// TIA Portal V18 export
FUNCTION "Pressure control" : Void   // FC24, LAD
{ S7_Optimized_Access := 'TRUE' }
VERSION : 0.1
// stored: AutoNumber true, IsIECCheckEnabled false, SetENOAutomatically false, UDAEnableTagReadback false
BEGIN

REGION Network 1 (SCL): Pump A pressure setting Inlet

   IF "Pressure sensor Pump Inlet A" < 32767 AND "Control".Pressure_sensor_select = 0 THEN
       "pressure".Misc."Pump A Scalx valueIN" := SCALE_X(MIN := 0.0,
                                                           VALUE := NORM_X(MIN := 0,
                                                                           VALUE := "Pressure sensor Pump Inlet A",
                                                                           MAX := 27648),
                                                           MAX := "pressure".A."pressure at 20mA");
   ELSIF "Pressure sensor Pump Inlet A_mA" < 32767 AND "Control".Pressure_sensor_select = 1 THEN
       "pressure".Misc."Pump A Scalx valueIN" := SCALE_X(MIN := 0.0,
                                                           VALUE := NORM_X(MIN := 0,
                                                                           VALUE := "Pressure sensor Pump Inlet A_mA",
                                                                           MAX := 27648),
                                                           MAX := "pressure".A."pressure at 20mA");
   END_IF;

   "Alarm_DB".input.alarm[15] := (("Control".Pressure_sensor_select = 0) AND ("Pressure sensor Pump Inlet A" >= 32767)) OR (("Control".Pressure_sensor_select = 1) AND ("Pressure sensor Pump Inlet A_mA" >= 32767));
END_REGION

REGION Network 2 (SCL): Pump A pressure setting Outlet

   IF "Pressure Sensor Pump Outlet A" < 32767 THEN
       "pressure".Misc."Pump A Scalx valueOUT" := SCALE_X(MIN := 0.0,
                                                           VALUE := NORM_X(MIN := 0,
                                                                           VALUE := "Pressure Sensor Pump Outlet A",
                                                                           MAX := 27648),
                                                           MAX := "pressure".A_Outlet."pressure at 20mA");
   END_IF;
END_REGION

REGION Network 3: gear Pump A pressure
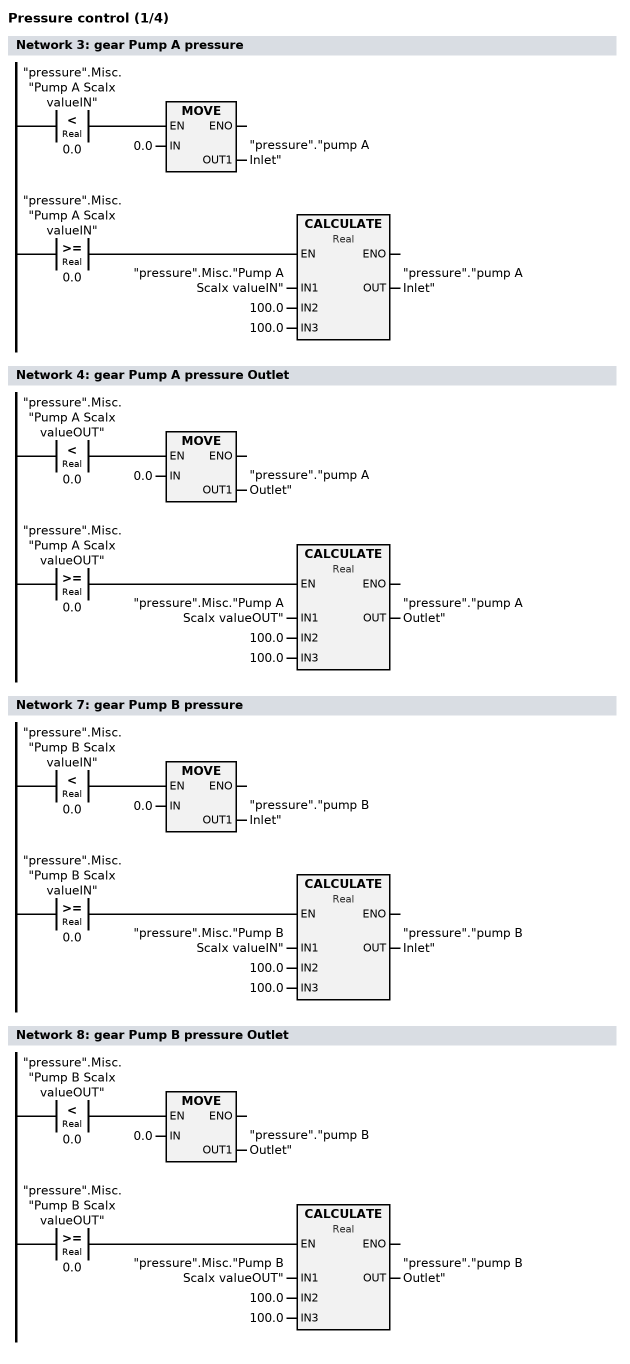
   RUNG wire#powerrail
      { S7_Templates := "SrcType := Real" } LT_Contact(in1 := "pressure".Misc."Pump A Scalx valueIN", in2 := 0.0)
      Move(in := 0.0, out1 => "pressure"."pump A Inlet")
   END_RUNG
   RUNG wire#powerrail
      { S7_Templates := "SrcType := Real" } GE_Contact(in1 := "pressure".Misc."Pump A Scalx valueIN", in2 := 0.0)
      { S7_Templates := "SrcType := Real"; S7_Expression := "ROUND(IN1*IN2)/IN3" } Calculate(in1 := "pressure".Misc."Pump A Scalx valueIN", in2 := 100.0, in3 := 100.0, out => "pressure"."pump A Inlet")
   END_RUNG
   // the same network as SCL:
   IF "pressure".Misc."Pump A Scalx valueIN" < 0.0 THEN "pressure"."pump A Inlet" := 0.0; END_IF;
   IF "pressure".Misc."Pump A Scalx valueIN" >= 0.0 THEN
       "pressure"."pump A Inlet" := ROUND("pressure".Misc."Pump A Scalx valueIN"*100.0)/100.0;
   END_IF;
END_REGION

REGION Network 4: gear Pump A pressure Outlet
   RUNG wire#powerrail
      { S7_Templates := "SrcType := Real" } LT_Contact(in1 := "pressure".Misc."Pump A Scalx valueOUT", in2 := 0.0)
      Move(in := 0.0, out1 => "pressure"."pump A Outlet")
   END_RUNG
   RUNG wire#powerrail
      { S7_Templates := "SrcType := Real" } GE_Contact(in1 := "pressure".Misc."Pump A Scalx valueOUT", in2 := 0.0)
      { S7_Templates := "SrcType := Real"; S7_Expression := "ROUND(IN1*IN2)/IN3" } Calculate(in1 := "pressure".Misc."Pump A Scalx valueOUT", in2 := 100.0, in3 := 100.0, out => "pressure"."pump A Outlet")
   END_RUNG
   // the same network as SCL:
   IF "pressure".Misc."Pump A Scalx valueOUT" < 0.0 THEN "pressure"."pump A Outlet" := 0.0; END_IF;
   IF "pressure".Misc."Pump A Scalx valueOUT" >= 0.0 THEN
       "pressure"."pump A Outlet" := ROUND("pressure".Misc."Pump A Scalx valueOUT"*100.0)/100.0;
   END_IF;
END_REGION

REGION Network 5 (SCL): Pump b pressure setting Inlet

   IF "Pressure Sensor Pump Inlet B" < 32767 AND "Control".Pressure_sensor_select = 0 THEN
       "pressure".Misc."Pump B Scalx valueIN" := SCALE_X(MIN := 0.0,
                                                           VALUE := NORM_X(MIN := 0,
                                                                           VALUE := "Pressure Sensor Pump Inlet B",
                                                                           MAX := 27648),
                                                           MAX := "pressure".B."pressure at 20mA");
   ELSIF "Pressure Sensor Pump Inlet B_mA" < 32767 AND "Control".Pressure_sensor_select = 1 THEN
       "pressure".Misc."Pump B Scalx valueIN" := SCALE_X(MIN := 0.0,
                                                           VALUE := NORM_X(MIN := 0,
                                                                           VALUE := "Pressure Sensor Pump Inlet B_mA",
                                                                           MAX := 27648),
                                                           MAX := "pressure".B."pressure at 20mA");
   END_IF;
   "Alarm_DB".input.alarm[0] := (("Control".Pressure_sensor_select = 0) AND ("Pressure Sensor Pump Inlet B" >= 32767)) OR (("Control".Pressure_sensor_select = 1) AND ("Pressure Sensor Pump Inlet B_mA" >= 32767));
END_REGION

REGION Network 6 (SCL): Pump b pressure setting Outlet

   IF "Pressure Sensor Pump Outlet B" < 32767 THEN
       "pressure".Misc."Pump B Scalx valueOUT" := SCALE_X(MIN := 0.0,
                                                           VALUE := NORM_X(MIN := 0,
                                                                           VALUE := "Pressure Sensor Pump Outlet B",
                                                                           MAX := 27648),
                                                           MAX := "pressure".B_Outlet."pressure at 20mA");
   END_IF;
END_REGION

REGION Network 7: gear Pump B pressure
   RUNG wire#powerrail
      { S7_Templates := "SrcType := Real" } LT_Contact(in1 := "pressure".Misc."Pump B Scalx valueIN", in2 := 0.0)
      Move(in := 0.0, out1 => "pressure"."pump B Inlet")
   END_RUNG
   RUNG wire#powerrail
      { S7_Templates := "SrcType := Real" } GE_Contact(in1 := "pressure".Misc."Pump B Scalx valueIN", in2 := 0.0)
      { S7_Templates := "SrcType := Real"; S7_Expression := "ROUND(IN1*IN2)/IN3" } Calculate(in1 := "pressure".Misc."Pump B Scalx valueIN", in2 := 100.0, in3 := 100.0, out => "pressure"."pump B Inlet")
   END_RUNG
   // the same network as SCL:
   IF "pressure".Misc."Pump B Scalx valueIN" < 0.0 THEN "pressure"."pump B Inlet" := 0.0; END_IF;
   IF "pressure".Misc."Pump B Scalx valueIN" >= 0.0 THEN
       "pressure"."pump B Inlet" := ROUND("pressure".Misc."Pump B Scalx valueIN"*100.0)/100.0;
   END_IF;
END_REGION

REGION Network 8: gear Pump B pressure Outlet
   RUNG wire#powerrail
      { S7_Templates := "SrcType := Real" } LT_Contact(in1 := "pressure".Misc."Pump B Scalx valueOUT", in2 := 0.0)
      Move(in := 0.0, out1 => "pressure"."pump B Outlet")
   END_RUNG
   RUNG wire#powerrail
      { S7_Templates := "SrcType := Real" } GE_Contact(in1 := "pressure".Misc."Pump B Scalx valueOUT", in2 := 0.0)
      { S7_Templates := "SrcType := Real"; S7_Expression := "ROUND(IN1*IN2)/IN3" } Calculate(in1 := "pressure".Misc."Pump B Scalx valueOUT", in2 := 100.0, in3 := 100.0, out => "pressure"."pump B Outlet")
   END_RUNG
   // the same network as SCL:
   IF "pressure".Misc."Pump B Scalx valueOUT" < 0.0 THEN "pressure"."pump B Outlet" := 0.0; END_IF;
   IF "pressure".Misc."Pump B Scalx valueOUT" >= 0.0 THEN
       "pressure"."pump B Outlet" := ROUND("pressure".Misc."Pump B Scalx valueOUT"*100.0)/100.0;
   END_IF;
END_REGION

REGION Network 9: mbar to bar
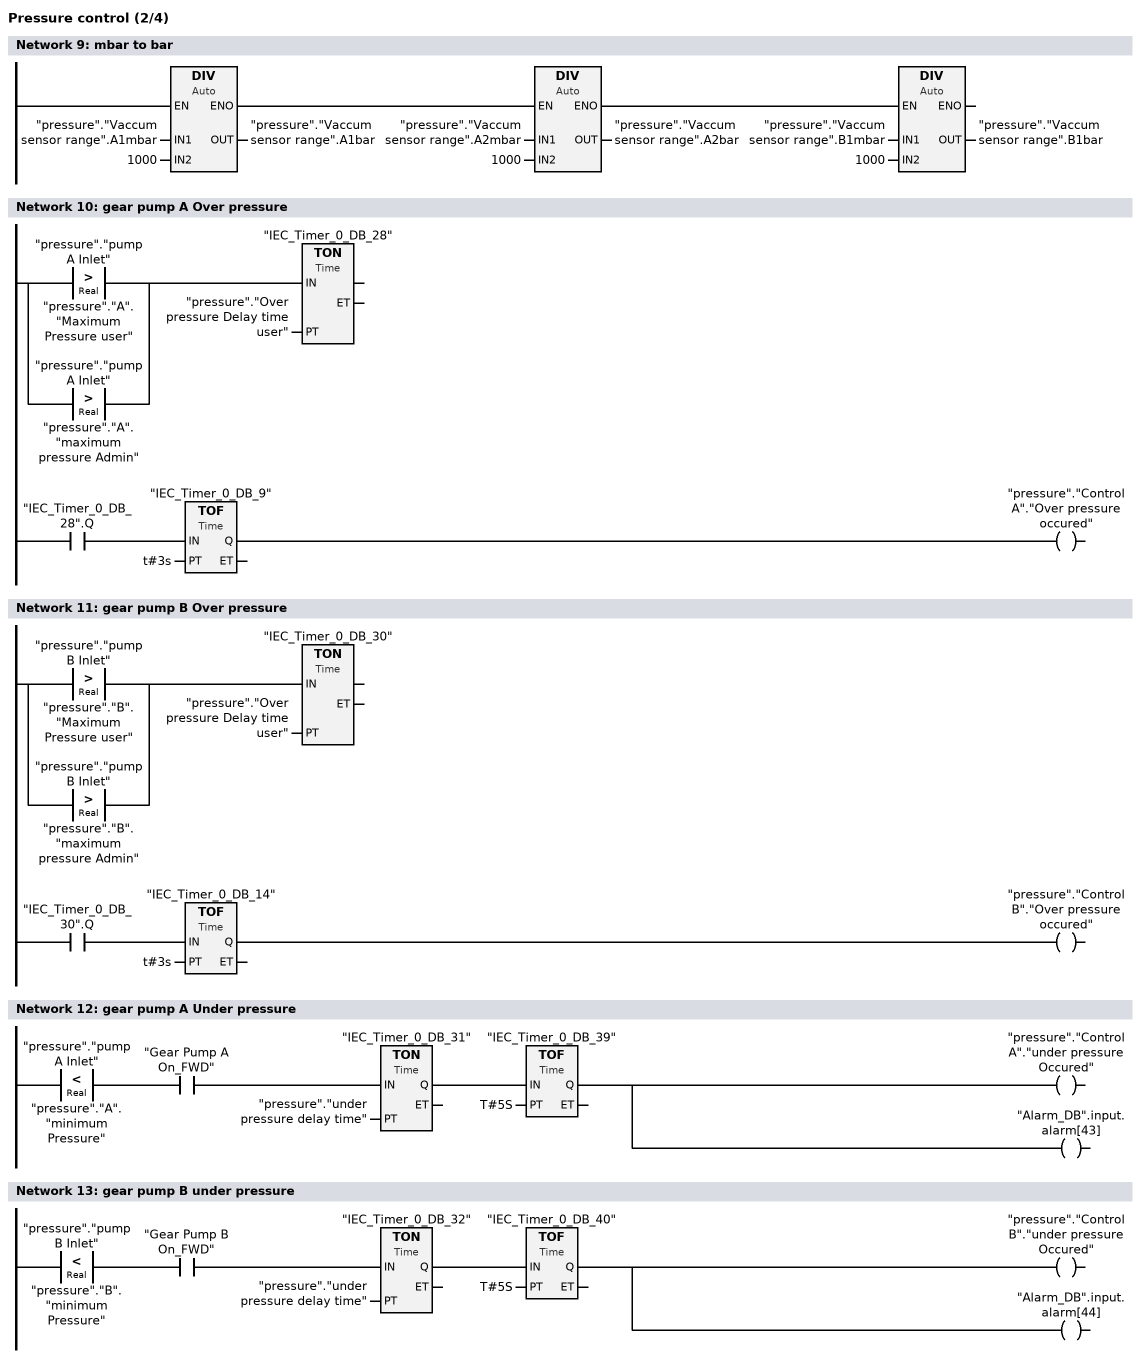
   RUNG wire#powerrail
      Div(in1 := "pressure"."Vaccum  sensor range".A1mbar, in2 := 1000, out => "pressure"."Vaccum  sensor range".A1bar)
      Div(in1 := "pressure"."Vaccum  sensor range".A2mbar, in2 := 1000, out => "pressure"."Vaccum  sensor range".A2bar)
      Div(in1 := "pressure"."Vaccum  sensor range".B1mbar, in2 := 1000, out => "pressure"."Vaccum  sensor range".B1bar)
   END_RUNG
   // the same network as SCL:
   "pressure"."Vaccum  sensor range".A1bar := "pressure"."Vaccum  sensor range".A1mbar / 1000;
   "pressure"."Vaccum  sensor range".A2bar := "pressure"."Vaccum  sensor range".A2mbar / 1000;
   "pressure"."Vaccum  sensor range".B1bar := "pressure"."Vaccum  sensor range".B1mbar / 1000;
END_REGION

REGION Network 10: gear pump A Over pressure
   RUNG wire#powerrail
      { S7_Templates := "SrcType := Real" } GT_Contact(in1 := "pressure"."pump A Inlet", in2 := "pressure"."A"."Maximum Pressure user")
      wire#w1
      { S7_Templates := "time_type := Time" } "IEC_Timer_0_DB_28".TON(pt := "pressure"."Over pressure Delay time user", et =>)
   END_RUNG
   RUNG wire#powerrail
      { S7_Templates := "SrcType := Real" } GT_Contact(in1 := "pressure"."pump A Inlet", in2 := "pressure"."A"."maximum pressure Admin")
   END_RUNG wire#w1
   RUNG wire#powerrail
      Contact( "IEC_Timer_0_DB_28".Q )
      { S7_Templates := "time_type := Time" } "IEC_Timer_0_DB_9".TOF(pt := t#3s, et =>)
      Coil( "pressure"."Control A"."Over pressure occured" )
   END_RUNG
   // the same network as SCL:
   "IEC_Timer_0_DB_28".TON(IN := ("pressure"."pump A Inlet" > "pressure"."A"."Maximum Pressure user") OR ("pressure"."pump A Inlet" > "pressure"."A"."maximum pressure Admin"),
                           PT := "pressure"."Over pressure Delay time user");
   "IEC_Timer_0_DB_9".TOF(IN := "IEC_Timer_0_DB_28".Q, PT := t#3s);
   "pressure"."Control A"."Over pressure occured" := "IEC_Timer_0_DB_9".Q;
END_REGION

REGION Network 11: gear pump B Over pressure
   RUNG wire#powerrail
      { S7_Templates := "SrcType := Real" } GT_Contact(in1 := "pressure"."pump B Inlet", in2 := "pressure"."B"."Maximum Pressure user")
      wire#w1
      { S7_Templates := "time_type := Time" } "IEC_Timer_0_DB_30".TON(pt := "pressure"."Over pressure Delay time user", et =>)
   END_RUNG
   RUNG wire#powerrail
      { S7_Templates := "SrcType := Real" } GT_Contact(in1 := "pressure"."pump B Inlet", in2 := "pressure"."B"."maximum pressure Admin")
   END_RUNG wire#w1
   RUNG wire#powerrail
      Contact( "IEC_Timer_0_DB_30".Q )
      { S7_Templates := "time_type := Time" } "IEC_Timer_0_DB_14".TOF(pt := t#3s, et =>)
      Coil( "pressure"."Control B"."Over pressure occured" )
   END_RUNG
   // the same network as SCL:
   "IEC_Timer_0_DB_30".TON(IN := ("pressure"."pump B Inlet" > "pressure"."B"."Maximum Pressure user") OR ("pressure"."pump B Inlet" > "pressure"."B"."maximum pressure Admin"),
                           PT := "pressure"."Over pressure Delay time user");
   "IEC_Timer_0_DB_14".TOF(IN := "IEC_Timer_0_DB_30".Q, PT := t#3s);
   "pressure"."Control B"."Over pressure occured" := "IEC_Timer_0_DB_14".Q;
END_REGION

REGION Network 12: gear pump A Under pressure
   RUNG wire#powerrail
      { S7_Templates := "SrcType := Real" } LT_Contact(in1 := "pressure"."pump A Inlet", in2 := "pressure"."A"."minimum Pressure")
      Contact( "Gear Pump A On_FWD" )
      { S7_Templates := "time_type := Time" } "IEC_Timer_0_DB_31".TON(pt := "pressure"."under pressure delay time", et =>)
      { S7_Templates := "time_type := Time" } "IEC_Timer_0_DB_39".TOF(pt := T#5S, et =>)
      wire#w1
      Coil( "pressure"."Control A"."under pressure Occured" )
   END_RUNG
   RUNG wire#w1
      Coil( "Alarm_DB".input.alarm[43] )
   END_RUNG
   // the same network as SCL:
   "IEC_Timer_0_DB_31".TON(IN := ("pressure"."pump A Inlet" < "pressure"."A"."minimum Pressure") AND "Gear Pump A On_FWD",
                           PT := "pressure"."under pressure delay time");
   "IEC_Timer_0_DB_39".TOF(IN := "IEC_Timer_0_DB_31".Q, PT := T#5S);
   "pressure"."Control A"."under pressure Occured" := "IEC_Timer_0_DB_39".Q;
   "Alarm_DB".input.alarm[43] := "IEC_Timer_0_DB_39".Q;
END_REGION

REGION Network 13: gear pump B under pressure
   RUNG wire#powerrail
      { S7_Templates := "SrcType := Real" } LT_Contact(in1 := "pressure"."pump B Inlet", in2 := "pressure"."B"."minimum Pressure")
      Contact( "Gear Pump B On_FWD" )
      { S7_Templates := "time_type := Time" } "IEC_Timer_0_DB_32".TON(pt := "pressure"."under pressure delay time", et =>)
      { S7_Templates := "time_type := Time" } "IEC_Timer_0_DB_40".TOF(pt := T#5S, et =>)
      wire#w1
      Coil( "pressure"."Control B"."under pressure Occured" )
   END_RUNG
   RUNG wire#w1
      Coil( "Alarm_DB".input.alarm[44] )
   END_RUNG
   // the same network as SCL:
   "IEC_Timer_0_DB_32".TON(IN := ("pressure"."pump B Inlet" < "pressure"."B"."minimum Pressure") AND "Gear Pump B On_FWD",
                           PT := "pressure"."under pressure delay time");
   "IEC_Timer_0_DB_40".TOF(IN := "IEC_Timer_0_DB_32".Q, PT := T#5S);
   "pressure"."Control B"."under pressure Occured" := "IEC_Timer_0_DB_40".Q;
   "Alarm_DB".input.alarm[44] := "IEC_Timer_0_DB_40".Q;
END_REGION

REGION Network 14: gear pump A Over pressure outlet
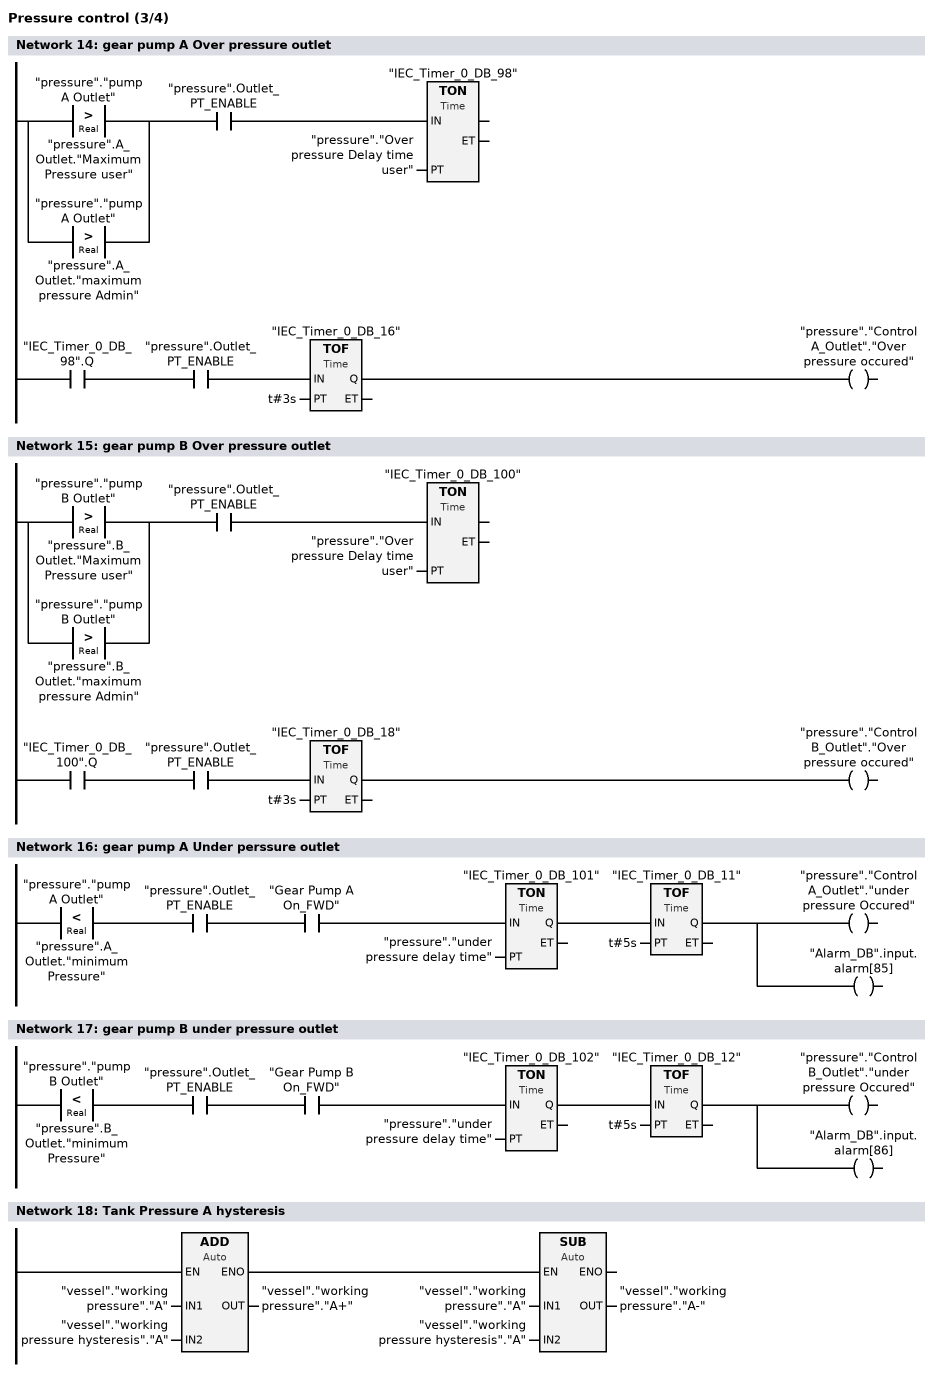
   RUNG wire#powerrail
      { S7_Templates := "SrcType := Real" } GT_Contact(in1 := "pressure"."pump A Outlet", in2 := "pressure".A_Outlet."Maximum Pressure user")
      wire#w1
      Contact( "pressure".Outlet_PT_ENABLE )
      { S7_Templates := "time_type := Time" } "IEC_Timer_0_DB_98".TON(pt := "pressure"."Over pressure Delay time user", et =>)
   END_RUNG
   RUNG wire#powerrail
      { S7_Templates := "SrcType := Real" } GT_Contact(in1 := "pressure"."pump A Outlet", in2 := "pressure".A_Outlet."maximum pressure Admin")
   END_RUNG wire#w1
   RUNG wire#powerrail
      Contact( "IEC_Timer_0_DB_98".Q )
      Contact( "pressure".Outlet_PT_ENABLE )
      { S7_Templates := "time_type := Time" } "IEC_Timer_0_DB_16".TOF(pt := t#3s, et =>)
      Coil( "pressure"."Control A_Outlet"."Over pressure occured" )
   END_RUNG
   // the same network as SCL:
   "IEC_Timer_0_DB_98".TON(IN := (("pressure"."pump A Outlet" > "pressure".A_Outlet."Maximum Pressure user") OR ("pressure"."pump A Outlet" > "pressure".A_Outlet."maximum pressure Admin")) AND "pressure".Outlet_PT_ENABLE,
                           PT := "pressure"."Over pressure Delay time user");
   "IEC_Timer_0_DB_16".TOF(IN := "IEC_Timer_0_DB_98".Q AND "pressure".Outlet_PT_ENABLE, PT := t#3s);
   "pressure"."Control A_Outlet"."Over pressure occured" := "IEC_Timer_0_DB_16".Q;
END_REGION

REGION Network 15: gear pump B Over pressure outlet
   RUNG wire#powerrail
      { S7_Templates := "SrcType := Real" } GT_Contact(in1 := "pressure"."pump B Outlet", in2 := "pressure".B_Outlet."Maximum Pressure user")
      wire#w1
      Contact( "pressure".Outlet_PT_ENABLE )
      { S7_Templates := "time_type := Time" } "IEC_Timer_0_DB_100".TON(pt := "pressure"."Over pressure Delay time user", et =>)
   END_RUNG
   RUNG wire#powerrail
      { S7_Templates := "SrcType := Real" } GT_Contact(in1 := "pressure"."pump B Outlet", in2 := "pressure".B_Outlet."maximum pressure Admin")
   END_RUNG wire#w1
   RUNG wire#powerrail
      Contact( "IEC_Timer_0_DB_100".Q )
      Contact( "pressure".Outlet_PT_ENABLE )
      { S7_Templates := "time_type := Time" } "IEC_Timer_0_DB_18".TOF(pt := t#3s, et =>)
      Coil( "pressure"."Control B_Outlet"."Over pressure occured" )
   END_RUNG
   // the same network as SCL:
   "IEC_Timer_0_DB_100".TON(IN := (("pressure"."pump B Outlet" > "pressure".B_Outlet."Maximum Pressure user") OR ("pressure"."pump B Outlet" > "pressure".B_Outlet."maximum pressure Admin")) AND "pressure".Outlet_PT_ENABLE,
                           PT := "pressure"."Over pressure Delay time user");
   "IEC_Timer_0_DB_18".TOF(IN := "IEC_Timer_0_DB_100".Q AND "pressure".Outlet_PT_ENABLE, PT := t#3s);
   "pressure"."Control B_Outlet"."Over pressure occured" := "IEC_Timer_0_DB_18".Q;
END_REGION

REGION Network 16: gear pump A Under perssure outlet
   RUNG wire#powerrail
      { S7_Templates := "SrcType := Real" } LT_Contact(in1 := "pressure"."pump A Outlet", in2 := "pressure".A_Outlet."minimum Pressure")
      Contact( "pressure".Outlet_PT_ENABLE )
      Contact( "Gear Pump A On_FWD" )
      { S7_Templates := "time_type := Time" } "IEC_Timer_0_DB_101".TON(pt := "pressure"."under pressure delay time", et =>)
      { S7_Templates := "time_type := Time" } "IEC_Timer_0_DB_11".TOF(pt := t#5s, et =>)
      wire#w1
      Coil( "pressure"."Control A_Outlet"."under pressure Occured" )
   END_RUNG
   RUNG wire#w1
      Coil( "Alarm_DB".input.alarm[85] )
   END_RUNG
   // the same network as SCL:
   "IEC_Timer_0_DB_101".TON(IN := ("pressure"."pump A Outlet" < "pressure".A_Outlet."minimum Pressure") AND "pressure".Outlet_PT_ENABLE AND "Gear Pump A On_FWD",
                           PT := "pressure"."under pressure delay time");
   "IEC_Timer_0_DB_11".TOF(IN := "IEC_Timer_0_DB_101".Q, PT := t#5s);
   "pressure"."Control A_Outlet"."under pressure Occured" := "IEC_Timer_0_DB_11".Q;
   "Alarm_DB".input.alarm[85] := "IEC_Timer_0_DB_11".Q;
END_REGION

REGION Network 17: gear pump B under pressure outlet
   RUNG wire#powerrail
      { S7_Templates := "SrcType := Real" } LT_Contact(in1 := "pressure"."pump B Outlet", in2 := "pressure".B_Outlet."minimum Pressure")
      Contact( "pressure".Outlet_PT_ENABLE )
      Contact( "Gear Pump B On_FWD" )
      { S7_Templates := "time_type := Time" } "IEC_Timer_0_DB_102".TON(pt := "pressure"."under pressure delay time", et =>)
      { S7_Templates := "time_type := Time" } "IEC_Timer_0_DB_12".TOF(pt := t#5s, et =>)
      wire#w1
      Coil( "pressure"."Control B_Outlet"."under pressure Occured" )
   END_RUNG
   RUNG wire#w1
      Coil( "Alarm_DB".input.alarm[86] )
   END_RUNG
   // the same network as SCL:
   "IEC_Timer_0_DB_102".TON(IN := ("pressure"."pump B Outlet" < "pressure".B_Outlet."minimum Pressure") AND "pressure".Outlet_PT_ENABLE AND "Gear Pump B On_FWD",
                           PT := "pressure"."under pressure delay time");
   "IEC_Timer_0_DB_12".TOF(IN := "IEC_Timer_0_DB_102".Q, PT := t#5s);
   "pressure"."Control B_Outlet"."under pressure Occured" := "IEC_Timer_0_DB_12".Q;
   "Alarm_DB".input.alarm[86] := "IEC_Timer_0_DB_12".Q;
END_REGION

REGION Network 18: Tank Pressure A hysteresis
   RUNG wire#powerrail
      Add(in1 := "vessel"."working pressure"."A", in2 := "vessel"."working pressure hysteresis"."A", out => "vessel"."working pressure"."A+")
      Sub(in1 := "vessel"."working pressure"."A", in2 := "vessel"."working pressure hysteresis"."A", out => "vessel"."working pressure"."A-")
   END_RUNG
   // the same network as SCL:
   "vessel"."working pressure"."A+" := "vessel"."working pressure"."A" + "vessel"."working pressure hysteresis"."A";
   "vessel"."working pressure"."A-" := "vessel"."working pressure"."A" - "vessel"."working pressure hysteresis"."A";
END_REGION

REGION Network 19: Tank Pressure B hysteresis
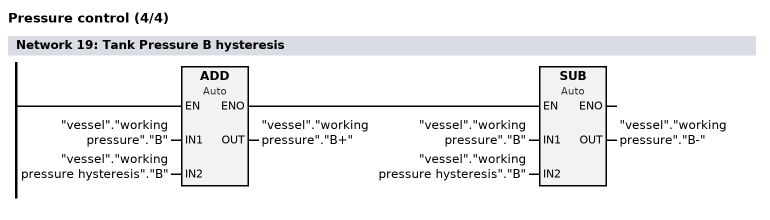
   RUNG wire#powerrail
      Add(in1 := "vessel"."working pressure"."B", in2 := "vessel"."working pressure hysteresis"."B", out => "vessel"."working pressure"."B+")
      Sub(in1 := "vessel"."working pressure"."B", in2 := "vessel"."working pressure hysteresis"."B", out => "vessel"."working pressure"."B-")
   END_RUNG
   // the same network as SCL:
   "vessel"."working pressure"."B+" := "vessel"."working pressure"."B" + "vessel"."working pressure hysteresis"."B";
   "vessel"."working pressure"."B-" := "vessel"."working pressure"."B" - "vessel"."working pressure hysteresis"."B";
END_REGION
END_FUNCTION
